// TIA Portal V19 export
TYPE "type_teachPara_Interface"
// stored: Access Published
   STRUCT
      constraint : "type_teachPara_constraint";
      plastic : "type_teachPara_plastic";
      ngConveyor { S7_SetPoint := 'True'} : "type_teachPara_ngConveyor";
      trayTypeSelect { S7_SetPoint := 'True'} : "LEXCHANGETRAY_typeTraySpecification";
   END_STRUCT;
END_TYPE
